Yaskawa INFORM job: R2_W66-W67(-70,-90)AWOK.JBI

/JOB
//NAME R2_W66-W67(-70,-90)AWOK
///FOLDERNAME AWOK
//POS
///NPOS 41,41,0,3,0,0
///TOOL 0
///POSTYPE PULSE
///PULSE
C00000=135635,-24500,-41716,-31750,82638,-33791
C00001=121173,28136,37388,-9783,95382,-11090
C00002=121152,31888,45574,-9734,92313,-10856
C00003=121144,33601,49119,-9722,91029,-10759
C00004=121138,33809,50614,-9717,90226,-10699
C00005=121144,33601,49119,-9722,91029,-10759
C00006=121116,38922,55034,-9721,90132,-10699
C00007=121113,42028,58811,-9718,89413,-10644
C00008=121116,38922,55034,-9721,90132,-10699
C00009=120187,34889,50757,-9920,90573,-11044
C00010=119360,34923,50783,-10093,90475,-11313
C00011=120187,34889,50757,-9920,90573,-11044
C00012=120195,33129,47147,-9931,91873,-11144
C00013=120213,29283,38831,-9979,94971,-11386
C00014=124262,41791,46564,15679,81195,-12986
C00015=125301,47706,56682,15822,77923,-13043
C00016=125710,50402,61178,15901,76514,-13085
C00017=125721,50569,62633,15951,75732,-13184
C00018=125710,50402,61178,15901,76514,-13085
C00019=116694,23381,45616,38194,53668,-63001
C00020=116738,26176,48836,38432,53217,-63176
C00021=116694,23381,45616,38194,53668,-63001
C00022=118829,36803,52428,28844,69518,-21730
C00023=119649,36749,52382,28805,69244,-21478
C00024=118829,36803,52428,28844,69518,-21730
C00025=118147,34363,48669,28702,70681,-21695
C00026=116410,28824,40027,28425,73448,-21667
C00027=120722,36277,52307,-21922,60833,8108
C00028=120725,29599,36610,-20842,66654,6972
C00029=109986,44671,45472,-4739,72285,-39309
C00030=109829,25936,29329,-1019,58563,-75027
C00031=109063,18233,35812,1126,41708,-75508
C00032=120730,33890,48639,-21720,61795,7914
C00033=120725,33272,48739,-21793,61440,7984
C00034=141865,29563,45829,-7389,45625,-61280
C00035=141165,29364,46195,-1871,44021,-62157
C00036=141194,19904,22517,-1630,53727,-62321
C00037=141194,19904,22517,-1630,53727,-62321
C00038=132020,10447,-13346,2437,70990,-65718
C00039=130510,-84668,-101602,2499,71155,-65752
C00040=130510,-84668,-101602,2499,71155,-65752
BC00000=108350,311250,937615
BC00001=156279,84855,733616
BC00002=156279,84855,733616
BC00003=156279,84855,733616
BC00004=156279,84855,733616
BC00005=156279,84855,733616
BC00006=156279,84855,733616
BC00007=156279,84855,733616
BC00008=156279,84855,733616
BC00009=156279,84855,733616
BC00010=156279,84855,733616
BC00011=156279,84855,733616
BC00012=156279,84855,733616
BC00013=156279,84855,733616
BC00014=113113,130089,688648
BC00015=113113,130089,688648
BC00016=113113,130089,688648
BC00017=113113,130089,688648
BC00018=113113,130089,688648
BC00019=113113,130089,688648
BC00020=113113,130089,688648
BC00021=113113,130089,688648
BC00022=113113,130089,688648
BC00023=113113,130089,688648
BC00024=113113,130089,688648
BC00025=113113,130089,688648
BC00026=113113,130089,688648
BC00027=131179,148967,829365
BC00028=131601,148971,721839
BC00029=135449,142609,694419
BC00030=135449,142609,694419
BC00031=135449,142609,694419
BC00032=135449,142609,694419
BC00033=135449,142609,694419
BC00034=135448,142610,694416
BC00035=135448,142610,694416
BC00036=135448,142610,694416
BC00037=135448,142610,694416
BC00038=135448,142610,694416
BC00039=135448,142610,876221
BC00040=135448,299476,876221
///POSTYPE BASE
///RECTAN
///RCONF 0,0,0,0,0,0,0,0,0,0,0,0,0,0,0,0,0,0,0,0,0,0,0,0
P00006=0.222,-3.123,-1.508,0.0000,0.0000,0.0000
P00021=-0.225,-6.128,-0.405,0.0000,0.0000,0.0000
P00022=0.222,-3.123,-1.508,0.0000,0.0000,0.0000
//INST
///DATE 2023/11/16 10:49
///ATTR SC,RW
///GROUP1 RB1,BS1
NOP
'r2_W66-W67(-70,-90)
MOVJ C00000 BC00000 VJ=20.00
'Path S1112 (for W504)
SFTOF
MOVJ C00001 BC00001 VJ=20.00
MOVJ C00002 BC00002 VJ=20.00
MOVL C00003 BC00003 V=60.0
REFP 3 C00004 BC00004
CALL JOB:SEARCH-R1
SET P021 P006
SFTON P021
MOVL C00005 BC00005 V=60.0
MOVL C00006 BC00006 V=60.0
REFP 3 C00007 BC00007
CALL JOB:SEARCH-R1
SET P021 P006
SFTON P021
MOVL C00008 BC00008 V=60.0
MOVL C00009 BC00009 V=60.0
REFP 3 C00010 BC00010
CALL JOB:SEARCH-R1
SET P021 P006
SFTON P021
MOVL C00011 BC00011 V=60.0
MOVL C00012 BC00012 V=100.0
MOVL C00013 BC00013 V=100.0
'Path S1113 (for W504)
SFTOF
MOVJ C00014 BC00014 VJ=20.00
MOVJ C00015 BC00015 VJ=20.00
MOVL C00016 BC00016 V=60.0
REFP 3 C00017 BC00017
CALL JOB:SEARCH-R1
SET P022 P006
SFTON P022
MOVL C00018 BC00018 V=60.0
MOVL C00019 BC00019 V=60.0
REFP 3 C00020 BC00020
CALL JOB:SEARCH-R1
SET P022 P006
SFTON P022
MOVL C00021 BC00021 V=60.0
MOVL C00022 BC00022 V=60.0
REFP 3 C00023 BC00023
CALL JOB:SEARCH-R1
SET P022 P006
SFTON P022
MOVL C00024 BC00024 V=60.0
MOVL C00025 BC00025 V=100.0
MOVL C00026 BC00026 V=100.0
'Path W1114
SFTOF
SFTON P021
MOVJ C00027 BC00027 VJ=20.00
MOVJ C00028 BC00028 VJ=20.00
MOVJ C00029 BC00029 VJ=20.00
MOVJ C00030 BC00030 VJ=20.00
MOVL C00031 BC00031 V=100.0 PL=0
REFP 1 C00032 BC00032
REFP 2 C00033 BC00033
MACRO1 MJ#(0) ARGF9
ARCON
SFTOF
SFTON P022
MOVL C00034 BC00034 V=10.8
MOVL C00035 BC00035 V=10.8
ARCOF
MOVL C00036 BC00036 V=100.0
MOVL C00037 BC00037 V=100.0
MOVJ C00038 BC00038 VJ=20.00
MOVJ C00039 BC00039 VJ=20.00
MOVJ C00040 BC00040 VJ=20.00
END
